(* PLC project LibIT_MBRTU_MASTER, lamsystems-it.ru LibIT_MBRTU_MASTER 1 *)
(* stored: creationDateTime 2020-08-04T15:04:45, productRelease 0, modificationDateTime 2021-12-16T15:43:44, version 1 *)

(* ModBus RTU Master: Send Diagnostic Query *)
FUNCTION_BLOCK MbRtuDiag
  VAR_INPUT
    Ex : BOOL := FALSE;  (* allow exec. *)
    Mode : BOOL := FALSE;  (* work mode (0 - cicle exec 1 - single exec) *)
    Com : BYTE := 1;  (* number of COM-port *)
    ID : BYTE := 0;  (* ID of target device *)
    SubFunc : BYTE := 0;  (* sub code of ModBus function *)
    Num : BYTE := 1;  (* quantity of read registers *)
    I1 : WORD := 0;  (* transmit data byte 1 *)
    I2 : WORD := 0;  (* transmit data byte 2 *)
    I3 : WORD := 0;  (* transmit data byte 3 *)
    I4 : WORD := 0;  (* transmit data byte 4 *)
    I5 : WORD := 0;  (* transmit data byte 5 *)
    I6 : WORD := 0;  (* transmit data byte 6 *)
    I7 : WORD := 0;  (* transmit data byte 7 *)
    I8 : WORD := 0;  (* transmit data byte 8 *)
  END_VAR
  VAR_OUTPUT
    Ok : BYTE := 0;  (* code of result *)
    OutData : WORD := 0;  (* recive data byte 1 *)
  END_VAR
  VAR
    ExPrev : BOOL := FALSE;
  END_VAR

            {extern void AppMbRtuMaster_SendDiagQuery(MBRTUDIAG*);AppMbRtuMaster_SendDiagQuery(data__);}
          
END_FUNCTION_BLOCK

(* ModBus RTU Master: SET TOUT Value *)
FUNCTION_BLOCK MbRtuSetTimeOutValue
  VAR_INPUT
    Ex : BOOL := FALSE;  (* allow exec. *)
    Value : WORD := 500;  (* new timeout value *)
  END_VAR
  VAR_OUTPUT
    Ok : BYTE := 0;  (* code of result *)
  END_VAR
  VAR
    ExPrev : BOOL := FALSE;
  END_VAR

            {extern void AppMbRtuMaster_SetTimeOutValue(MBRTUSETTIMEOUTVALUE*);AppMbRtuMaster_SetTimeOutValue(data__);}
          
END_FUNCTION_BLOCK

(* ModBus RTU Master: GET TOUT Value *)
FUNCTION_BLOCK MbRtuGetTimeOutValue
  VAR_INPUT
    Ex : BOOL := FALSE;  (* allow exec. *)
  END_VAR
  VAR_OUTPUT
    Value : WORD := 500;  (* current timeout value *)
    Ok : BYTE := 0;  (* code of result *)
  END_VAR
  VAR
    ExPrev : BOOL := FALSE;
  END_VAR

            {extern void AppMbRtuMaster_GetTimeOutValue(MBRTUGETTIMEOUTVALUE*);AppMbRtuMaster_GetTimeOutValue(data__);}
          
END_FUNCTION_BLOCK

(* ModBus RTU Master: Read BOOL-registers *)
FUNCTION_BLOCK MbRtuReadBool
  VAR_INPUT
    Ex : BOOL := FALSE;  (* allow exec. *)
    Mode : BOOL := FALSE;  (* work mode (0 - cicle exec 1 - single exec) *)
    Com : BYTE := 1;  (* number of COM-port *)
    ID : BYTE := 0;  (* ID of target device *)
    Func : BYTE := 0;  (* code of ModBus function *)
    Addr1 : WORD := 0;  (* address of start register *)
    Num : BYTE := 1;  (* quantity of read registers *)
  END_VAR
  VAR_OUTPUT
    Ok : BYTE := 0;  (* code of result *)
    O1 : BOOL := FALSE;  (* register 1 *)
    O2 : BOOL := FALSE;  (* register 2 *)
    O3 : BOOL := FALSE;  (* register 3 *)
    O4 : BOOL := FALSE;  (* register 4 *)
    O5 : BOOL := FALSE;  (* register 5 *)
    O6 : BOOL := FALSE;  (* register 6 *)
    O7 : BOOL := FALSE;  (* register 7 *)
    O8 : BOOL := FALSE;  (* register 8 *)
  END_VAR
  VAR
    ExPrev : BOOL := FALSE;
  END_VAR

            {extern void AppMbRtuMaster_ReadBool(MBRTUREADBOOL*);AppMbRtuMaster_ReadBool(data__);}
          
END_FUNCTION_BLOCK

(* ModBus RTU Master: Read INT-registers *)
FUNCTION_BLOCK MbRtuReadInt
  VAR_INPUT
    Ex : BOOL := FALSE;  (* allow exec. *)
    Mode : BOOL := FALSE;  (* work mode (0 - cicle exec 1 - single exec) *)
    Com : BYTE := 1;  (* number of COM-port *)
    ID : BYTE := 0;  (* ID of target device *)
    Func : BYTE := 0;  (* code of ModBus function *)
    Addr1 : WORD := 0;  (* address of start register *)
    Num : BYTE := 1;  (* quantity of read registers *)
  END_VAR
  VAR_OUTPUT
    Ok : BYTE := 0;  (* code of result *)
    O1 : INT := 0;  (* register 1 *)
    O2 : INT := 0;  (* register 2 *)
    O3 : INT := 0;  (* register 3 *)
    O4 : INT := 0;  (* register 4 *)
    O5 : INT := 0;  (* register 5 *)
    O6 : INT := 0;  (* register 6 *)
    O7 : INT := 0;  (* register 7 *)
    O8 : INT := 0;  (* register 8 *)
  END_VAR
  VAR
    ExPrev : BOOL := FALSE;
  END_VAR

            {extern void AppMbRtuMaster_ReadInt(MBRTUREADINT*);AppMbRtuMaster_ReadInt(data__);}
          
END_FUNCTION_BLOCK

(* ModBus RTU Master: Read DINT-registers *)
FUNCTION_BLOCK MbRtuReadDInt
  VAR_INPUT
    Ex : BOOL := FALSE;  (* allow exec. *)
    Mode : BOOL := FALSE;  (* work mode (0 - cicle exec 1 - single exec) *)
    Com : BYTE := 1;  (* number of COM-port *)
    ID : BYTE := 0;  (* ID of target device *)
    Func : BYTE := 0;  (* code of ModBus function *)
    Addr1 : WORD := 0;  (* address of start register *)
    Num : BYTE := 1;  (* quantity of read registers *)
  END_VAR
  VAR_OUTPUT
    Ok : BYTE := 0;  (* code of result *)
    O1 : DINT := 0;  (* register 1 *)
    O2 : DINT := 0;  (* register 2 *)
    O3 : DINT := 0;  (* register 3 *)
    O4 : DINT := 0;  (* register 4 *)
    O5 : DINT := 0;  (* register 5 *)
    O6 : DINT := 0;  (* register 6 *)
    O7 : DINT := 0;  (* register 7 *)
    O8 : DINT := 0;  (* register 8 *)
  END_VAR
  VAR
    ExPrev : BOOL := FALSE;
  END_VAR

            {extern void AppMbRtuMaster_ReadDInt(MBRTUREADDINT*);AppMbRtuMaster_ReadDInt(data__);}
          
END_FUNCTION_BLOCK

(* ModBus RTU Master: Read WORD-registers *)
FUNCTION_BLOCK MbRtuReadWord
  VAR_INPUT
    Ex : BOOL := FALSE;  (* allow exec. *)
    Mode : BOOL := FALSE;  (* work mode (0 - cicle exec 1 - single exec) *)
    Com : BYTE := 1;  (* number of COM-port *)
    ID : BYTE := 0;  (* ID of target device *)
    Func : BYTE := 0;  (* code of ModBus function *)
    Addr1 : WORD := 0;  (* address of start register *)
    Num : BYTE := 1;  (* quantity of read registers *)
  END_VAR
  VAR_OUTPUT
    Ok : BYTE := 0;  (* code of result *)
    O1 : WORD := 0;  (* register 1 *)
    O2 : WORD := 0;  (* register 2 *)
    O3 : WORD := 0;  (* register 3 *)
    O4 : WORD := 0;  (* register 4 *)
    O5 : WORD := 0;  (* register 5 *)
    O6 : WORD := 0;  (* register 6 *)
    O7 : WORD := 0;  (* register 7 *)
    O8 : WORD := 0;  (* register 8 *)
  END_VAR
  VAR
    ExPrev : BOOL := FALSE;
  END_VAR

            {extern void AppMbRtuMaster_ReadWord(MBRTUREADWORD*);AppMbRtuMaster_ReadWord(data__);}
          
END_FUNCTION_BLOCK

(* ModBus RTU Master: Read DWORD-registers *)
FUNCTION_BLOCK MbRtuReadDWord
  VAR_INPUT
    Ex : BOOL := FALSE;  (* allow exec. *)
    Mode : BOOL := FALSE;  (* work mode (0 - cicle exec 1 - single exec) *)
    Com : BYTE := 1;  (* number of COM-port *)
    ID : BYTE := 0;  (* ID of target device *)
    Func : BYTE := 0;  (* code of ModBus function *)
    Addr1 : WORD := 0;  (* address of start register *)
    Num : BYTE := 1;  (* quantity of read registers *)
  END_VAR
  VAR_OUTPUT
    Ok : BYTE := 0;  (* code of result *)
    O1 : DWORD := 0;  (* register 1 *)
    O2 : DWORD := 0;  (* register 2 *)
    O3 : DWORD := 0;  (* register 3 *)
    O4 : DWORD := 0;  (* register 4 *)
    O5 : DWORD := 0;  (* register 5 *)
    O6 : DWORD := 0;  (* register 6 *)
    O7 : DWORD := 0;  (* register 7 *)
    O8 : DWORD := 0;  (* register 8 *)
  END_VAR
  VAR
    ExPrev : BOOL := FALSE;
  END_VAR

            {extern void AppMbRtuMaster_ReadDWord(MBRTUREADDWORD*);AppMbRtuMaster_ReadDWord(data__);}
          
END_FUNCTION_BLOCK

(* ModBus RTU Master: Read REAL-registers *)
FUNCTION_BLOCK MbRtuReadReal
  VAR_INPUT
    Ex : BOOL := FALSE;  (* allow exec. *)
    Mode : BOOL := FALSE;  (* work mode (0 - cicle exec 1 - single exec) *)
    Com : BYTE := 1;  (* number of COM-port *)
    ID : BYTE := 0;  (* ID of target device *)
    Func : BYTE := 0;  (* code of ModBus function *)
    Addr1 : WORD := 0;  (* address of start register *)
    Num : BYTE := 1;  (* quantity of read registers *)
  END_VAR
  VAR_OUTPUT
    Ok : BYTE := 0;  (* code of result *)
    O1 : REAL := 0.0;  (* register 1 *)
    O2 : REAL := 0.0;  (* register 2 *)
    O3 : REAL := 0.0;  (* register 3 *)
    O4 : REAL := 0.0;  (* register 4 *)
    O5 : REAL := 0.0;  (* register 5 *)
    O6 : REAL := 0.0;  (* register 6 *)
    O7 : REAL := 0.0;  (* register 7 *)
    O8 : REAL := 0.0;  (* register 8 *)
  END_VAR
  VAR
    ExPrev : BOOL := FALSE;
  END_VAR

            {extern void AppMbRtuMaster_ReadReal(MBRTUREADREAL*);AppMbRtuMaster_ReadReal(data__);}
          
END_FUNCTION_BLOCK

(* ModBus RTU Master: Write BOOL-registers *)
FUNCTION_BLOCK MbRtuWriteBool
  VAR_INPUT
    Ex : BOOL := FALSE;  (* allow exec. *)
    Mode : BOOL := FALSE;  (* work mode (0 - cicle exec 1 - single exec) *)
    Com : BYTE := 1;  (* number of COM-port *)
    ID : BYTE := 0;  (* ID of target device *)
    Func : BYTE := 0;  (* code of ModBus function *)
    Addr1 : WORD := 0;  (* address of start register *)
    Num : BYTE := 1;  (* quantity of write registers *)
    I1 : BOOL := FALSE;  (* register 1 *)
    I2 : BOOL := FALSE;  (* register 2 *)
    I3 : BOOL := FALSE;  (* register 3 *)
    I4 : BOOL := FALSE;  (* register 4 *)
    I5 : BOOL := FALSE;  (* register 5 *)
    I6 : BOOL := FALSE;  (* register 6 *)
    I7 : BOOL := FALSE;  (* register 7 *)
    I8 : BOOL := FALSE;  (* register 8 *)
  END_VAR
  VAR_OUTPUT
    Ok : BYTE := 0;  (* code of result *)
  END_VAR
  VAR
    ExPrev : BOOL := FALSE;
  END_VAR

            {extern void AppMbRtuMaster_WriteBool(MBRTUWRITEBOOL*);AppMbRtuMaster_WriteBool(data__);}
          
END_FUNCTION_BLOCK

(* ModBus RTU Master: Write INT-registers *)
FUNCTION_BLOCK MbRtuWriteInt
  VAR_INPUT
    Ex : BOOL := FALSE;  (* allow exec. *)
    Mode : BOOL := FALSE;  (* work mode (0 - cicle exec 1 - single exec) *)
    Com : BYTE := 1;  (* number of COM-port *)
    ID : BYTE := 0;  (* ID of target device *)
    Func : BYTE := 0;  (* code of ModBus function *)
    Addr1 : WORD := 0;  (* address of start register *)
    Num : BYTE := 1;  (* quantity of read registers *)
    I1 : INT := 0;  (* register 1 *)
    I2 : INT := 0;  (* register 2 *)
    I3 : INT := 0;  (* register 3 *)
    I4 : INT := 0;  (* register 4 *)
    I5 : INT := 0;  (* register 5 *)
    I6 : INT := 0;  (* register 6 *)
    I7 : INT := 0;  (* register 7 *)
    I8 : INT := 0;  (* register 8 *)
  END_VAR
  VAR_OUTPUT
    Ok : BYTE := 0;  (* code of result *)
  END_VAR
  VAR
    ExPrev : BOOL := FALSE;
  END_VAR

            {extern void AppMbRtuMaster_WriteInt(MBRTUWRITEINT*);AppMbRtuMaster_WriteInt(data__);}
          
END_FUNCTION_BLOCK

(* ModBus RTU Master: Write DINT-registers *)
FUNCTION_BLOCK MbRtuWriteDInt
  VAR_INPUT
    Ex : BOOL := FALSE;  (* allow exec. *)
    Mode : BOOL := FALSE;  (* work mode (0 - cicle exec 1 - single exec) *)
    Com : BYTE := 1;  (* number of COM-port *)
    ID : BYTE := 0;  (* ID of target device *)
    Func : BYTE := 0;  (* code of ModBus function *)
    Addr1 : WORD := 0;  (* address of start register *)
    Num : BYTE := 1;  (* quantity of read registers *)
    I1 : DINT := 0;  (* register 1 *)
    I2 : DINT := 0;  (* register 2 *)
    I3 : DINT := 0;  (* register 3 *)
    I4 : DINT := 0;  (* register 4 *)
    I5 : DINT := 0;  (* register 5 *)
    I6 : DINT := 0;  (* register 6 *)
    I7 : DINT := 0;  (* register 7 *)
    I8 : DINT := 0;  (* register 8 *)
  END_VAR
  VAR_OUTPUT
    Ok : BYTE := 0;  (* code of result *)
  END_VAR
  VAR
    ExPrev : BOOL := FALSE;
  END_VAR

            {extern void AppMbRtuMaster_WriteDInt(MBRTUWRITEDINT*);AppMbRtuMaster_WriteDInt(data__);}
          
END_FUNCTION_BLOCK

(* ModBus RTU Master: Write WORD-registers *)
FUNCTION_BLOCK MbRtuWriteWord
  VAR_INPUT
    Ex : BOOL := FALSE;  (* allow exec. *)
    Mode : BOOL := FALSE;  (* work mode (0 - cicle exec 1 - single exec) *)
    Com : BYTE := 1;  (* number of COM-port *)
    ID : BYTE := 0;  (* ID of target device *)
    Func : BYTE := 0;  (* code of ModBus function *)
    Addr1 : WORD := 0;  (* address of start register *)
    Num : BYTE := 1;  (* quantity of read registers *)
    I1 : WORD := 0;  (* register 1 *)
    I2 : WORD := 0;  (* register 2 *)
    I3 : WORD := 0;  (* register 3 *)
    I4 : WORD := 0;  (* register 4 *)
    I5 : WORD := 0;  (* register 5 *)
    I6 : WORD := 0;  (* register 6 *)
    I7 : WORD := 0;  (* register 7 *)
    I8 : WORD := 0;  (* register 8 *)
  END_VAR
  VAR_OUTPUT
    Ok : BYTE := 0;  (* code of result *)
  END_VAR
  VAR
    ExPrev : BOOL := FALSE;
  END_VAR

            {extern void AppMbRtuMaster_WriteWord(MBRTUWRITEWORD*);AppMbRtuMaster_WriteWord(data__);}
          
END_FUNCTION_BLOCK

(* ModBus RTU Master: Write DWORD-registers *)
FUNCTION_BLOCK MbRtuWriteDWord
  VAR_INPUT
    Ex : BOOL := FALSE;  (* allow exec. *)
    Mode : BOOL := FALSE;  (* work mode (0 - cicle exec 1 - single exec) *)
    Com : BYTE := 1;  (* number of COM-port *)
    ID : BYTE := 0;  (* ID of target device *)
    Func : BYTE := 0;  (* code of ModBus function *)
    Addr1 : WORD := 0;  (* address of start register *)
    Num : BYTE := 1;  (* quantity of read registers *)
    I1 : DWORD := 0;  (* register 1 *)
    I2 : DWORD := 0;  (* register 2 *)
    I3 : DWORD := 0;  (* register 3 *)
    I4 : DWORD := 0;  (* register 4 *)
    I5 : DWORD := 0;  (* register 5 *)
    I6 : DWORD := 0;  (* register 6 *)
    I7 : DWORD := 0;  (* register 7 *)
    I8 : DWORD := 0;  (* register 8 *)
  END_VAR
  VAR_OUTPUT
    Ok : BYTE := 0;  (* code of result *)
  END_VAR
  VAR
    ExPrev : BOOL := FALSE;
  END_VAR

            {extern void AppMbRtuMaster_WriteDWord(MBRTUWRITEDWORD*);AppMbRtuMaster_WriteDWord(data__);}
          
END_FUNCTION_BLOCK

(* ModBus RTU Master: Write REAL-registers *)
FUNCTION_BLOCK MbRtuWriteReal
  VAR_INPUT
    Ex : BOOL := FALSE;  (* allow exec. *)
    Mode : BOOL := FALSE;  (* work mode (0 - cicle exec 1 - single exec) *)
    Com : BYTE := 1;  (* number of COM-port *)
    ID : BYTE := 0;  (* ID of target device *)
    Func : BYTE := 0;  (* code of ModBus function *)
    Addr1 : WORD := 0;  (* address of start register *)
    Num : BYTE := 1;  (* quantity of read registers *)
    I1 : REAL := 0.0;  (* register 1 *)
    I2 : REAL := 0.0;  (* register 2 *)
    I3 : REAL := 0.0;  (* register 3 *)
    I4 : REAL := 0.0;  (* register 4 *)
    I5 : REAL := 0.0;  (* register 5 *)
    I6 : REAL := 0.0;  (* register 6 *)
    I7 : REAL := 0.0;  (* register 7 *)
    I8 : REAL := 0.0;  (* register 8 *)
  END_VAR
  VAR_OUTPUT
    Ok : BYTE := 0;  (* code of result *)
  END_VAR
  VAR
    ExPrev : BOOL := FALSE;
  END_VAR

            {extern void AppMbRtuMaster_WriteReal(MBRTUWRITEREAL*);AppMbRtuMaster_WriteReal(data__);}
          
END_FUNCTION_BLOCK
